RESOURCE_TYPE _CBCore2
  (* Standard: 61499-2 *)
  (* Version 0.1, 2019-00-29, hpea485, UOA *)
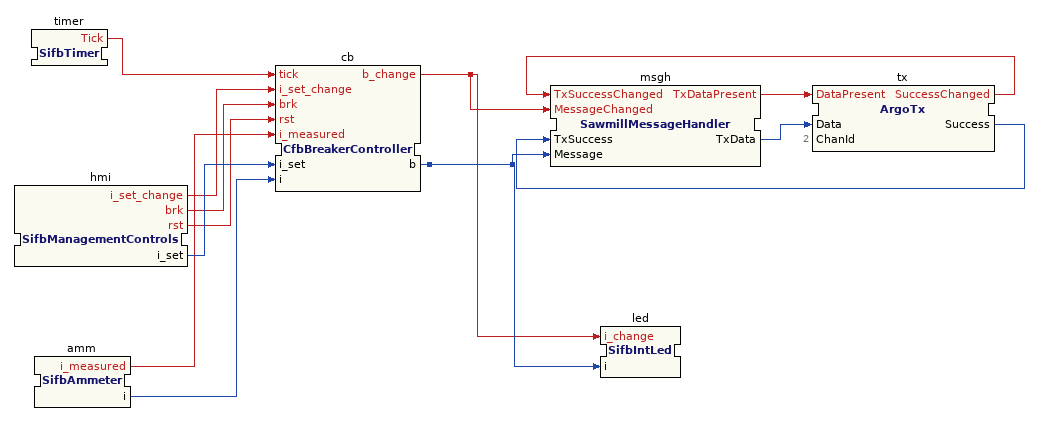
  FBS
    timer : SifbTimer;
    tx : ArgoTx(ChanId := 2);
    hmi : SifbManagementControls;
    led : SifbIntLed;
    cb : CfbBreakerController;
    amm : SifbAmmeter;
    msgh : SawmillMessageHandler;
  END_FBS
  EVENT_CONNECTIONS
    timer.Tick TO cb.tick;
    tx.SuccessChanged TO msgh.TxSuccessChanged;
    hmi.i_set_change TO cb.i_set_change;
    hmi.brk TO cb.brk;
    hmi.rst TO cb.rst;
    cb.b_change TO msgh.MessageChanged;
    cb.b_change TO led.i_change;
    amm.i_measured TO cb.i_measured;
    msgh.TxDataPresent TO tx.DataPresent;
  END_CONNECTIONS
  DATA_CONNECTIONS
    tx.Success TO msgh.TxSuccess;
    hmi.i_set TO cb.i_set;
    cb.b TO msgh.Message;
    cb.b TO led.i;
    amm.i TO cb.i;
    msgh.TxData TO tx.Data;
  END_CONNECTIONS
END_RESOURCE_TYPE
